TYPE InputBase_8311D824 :
STRUCT
END_STRUCT
END_TYPE

(* stored: Version 1.2.0.0, ProductVersion 3.1.4024.11
   DUT InputBase_8311D824: Id {47890048-2e31-4f57-80c8-c8b62539e236} *)
